// TIA Portal V16 export
// export: Created 2024-09-05T17:36:34.4302812Z, ExportSetting WithDefaults, DisplayName Totally Integrated Automation Portal, DisplayVersion V16 Update 6, DisplayName TIA Portal Version Control Interface, DisplayVersion V16 Update 2, DisplayName TIA Portal Openness, DisplayVersion V16 Update 6, DisplayName STEP 7 Professional, DisplayVersion V16 Update 6, DisplayName STEP 7 Safety, DisplayVersion V16, DisplayName WinCC Advanced, DisplayVersion V16 Update 6
VAR_GLOBAL   // PLC tag table "DM_FT"
   "DM_FT-TriggerEnable" AT %Q4.0 : Bool;
   "DM_FT-Trigger" AT %Q4.1 : Bool;
   "DM_FT-TriggerReady" AT %I4.0 : Bool;
   "DM_FT-TriggerAck" AT %I4.1 : Bool;
   "DM_FT-Acquiring" AT %I4.2 : Bool;
   "DM_FT-MissedAcq" AT %I4.3 : Bool;
   "DM_FT-TriggerID" AT %IW5 : Word;
   "DM_FT-BufferResultsEnable" AT %Q5.0 : Bool;
   "DM_FT-ResultsAck" AT %Q5.1 : Bool;
   "DM_FT-Decoding" AT %I7.0 : Bool;
   "DM_FT-Decode Complete" AT %I7.1 : Bool;
   "DM_FT-Results Buffer Overrun" AT %I7.2 : Bool;
   "DM_FT-Results Available" AT %I7.3 : Bool;
   "DM_FT-General Fault" AT %I7.7 : Bool;
   "DM_FT-Train Code" AT %Q6.0 : Bool;
   "DM_FT-Train Match String" AT %Q6.1 : Bool;
   "DM_FT-Train Focus" AT %Q6.2 : Bool;
   "DM_FT-Train Brightness" AT %Q6.3 : Bool;
   "DM_FT-Untrain" AT %Q6.4 : Bool;
   "DM_FT-Execute DMCC" AT %Q6.6 : Bool;
   "DM_FT-Set Match String" AT %Q6.7 : Bool;
   "DM_FT-Train Code Ack" AT %I8.0 : Bool;
   "DM_FT-Train Match String Ack" AT %I8.1 : Bool;
   "DM_FT-Train Focus Ack" AT %I8.2 : Bool;
   "DM_FT-Train Brightness Ack" AT %I8.3 : Bool;
   "DM_FT-Untrain Ack" AT %I8.4 : Bool;
   "DM_FT-Execute DMCC Ack" AT %I8.6 : Bool;
   "DM_FT-Set Match String Ack" AT %I8.7 : Bool;
   "DM_FT-UserData Option" AT %QW126 : Word;
   "DM_FT-UserData Length" AT %QW128 : Word;
   "DM_FT-UserData[0]" AT %QB130 : Byte;
   "DM_FT-UserData[1]" AT %QB131 : Byte;
   "DM_FT-UserData[2]" AT %QB132 : Byte;
   "DM_FT-UserData[3]" AT %QB133 : Byte;
   "DM_FT-UserData[4]" AT %QB134 : Byte;
   "DM_FT-UserData[5]" AT %QB135 : Byte;
   "DM_FT-UserData[6]" AT %QB136 : Byte;
   "DM_FT-UserData[7]" AT %QB137 : Byte;
   "DM_FT-UserData[8]" AT %QB138 : Byte;
   "DM_FT-UserData[9]" AT %QB139 : Byte;
   "DM_FT-UserData[10]" AT %QB140 : Byte;
   "DM_FT-UserData[11]" AT %QB141 : Byte;
   "DM_FT-UserData[12]" AT %QB142 : Byte;
   "DM_FT-UserData[13]" AT %QB143 : Byte;
   "DM_FT-UserData[14]" AT %QB144 : Byte;
   "DM_FT-UserData[15]" AT %QB145 : Byte;
   "DM_FT-ResultID" AT %IW126 : Word;
   "DM_FT-Result Code" AT %IW128 : Word;
   "DM_FT-Result Extended" AT %IW130 : Word;
   "DM_FT-Result Length" AT %IW132 : Word;
   "DM_FT-InspectionResults[0]" AT %IB134 : Byte;
   "DM_FT-InspectionResults[1]" AT %IB135 : Byte;
   "DM_FT-InspectionResults[2]" AT %IB136 : Byte;
   "DM_FT-InspectionResults[3]" AT %IB137 : Byte;
   "DM_FT-InspectionResults[4]" AT %IB138 : Byte;
   "DM_FT-InspectionResults[5]" AT %IB139 : Byte;
   "DM_FT-InspectionResults[6]" AT %IB140 : Byte;
   "DM_FT-InspectionResults[7]" AT %IB141 : Byte;
   "DM_FT-InspectionResults[8]" AT %IB142 : Byte;
   "DM_FT-InspectionResults[9]" AT %IB143 : Byte;
   "DM_FT-InspectionResults[10]" AT %IB144 : Byte;
   "DM_FT-InspectionResults[11]" AT %IB145 : Byte;
   "DM_FT-InspectionResults[12]" AT %IB146 : Byte;
   "DM_FT-InspectionResults[13]" AT %IB147 : Byte;
   "DM_FT-InspectionResults[14]" AT %IB148 : Byte;
   "DM_FT-InspectionResults[15]" AT %IB149 : Byte;
END_VAR
